PROGRAM StructuredText
VAR
	ChangeTime		:TIME:=T#1S;
	CountOnes		:INT:=1;
	CountFives		:INT:=1;
	JustOncePer 	:R_TRIG;
	DidSomething:BOOL;
	AlsoCountTo25	: BOOL;
END_VAR
VAR CONSTANT
	ST_DURATION	:TIME:=T#2S;
END_VAR

	Comparison_GVL.DefaultOFF	:=	Comparison_GVL.NormallyOpen_NO; //Sets DefaultOFF equal to whatever NormallyOpen is set to
	Comparison_GVL.DefaultON	:=	NOT Comparison_GVL.NormallyClosed_NC; //Sets DefaultON equal to the opposite of what NormallyClosed is set to
	
	Comparison_GVL.Tada			:= Comparison_GVL.This_And AND Comparison_GVL.And_This	AND NOT Comparison_GVL.But_NOT_This	AND
								(Comparison_GVL.This_Or OR Comparison_GVL.Or_This OR NOT Comparison_GVL.Or_NOT_This);
	
	// this line ^ and this next one technically do the same thing BUT if I wanted to do more complicated stuff or multiple things I need to use the IF 
	
	IF Comparison_GVL.This_And AND Comparison_GVL.And_This	AND NOT Comparison_GVL.But_NOT_This	AND
		(Comparison_GVL.This_Or OR Comparison_GVL.Or_This OR NOT Comparison_GVL.Or_NOT_This) THEN
		Comparison_GVL.Tada	:= TRUE;
	ELSE
		Comparison_GVL.Tada	:= FALSE;
	END_IF
	
	Comparison_GVL.OffTimer_TOF(IN:=Comparison_GVL.TurnOFFAfter,PT:= ST_DURATION);
	Comparison_GVL.OnTimer_TON(IN:=Comparison_GVL.TurnONAfter,PT:= ST_DURATION);
	Comparison_GVL.PulseTimer_TP(IN:=NOT Comparison_GVL.PulseTimer_TP.Q,PT:= ChangeTime);
	JustOncePer(CLK:= Comparison_GVL.PulseTimer_TP.Q);
	
	IF JustOncePer.Q THEN
		CountOnes:= CountOnes+1;
		Comparison_GVL.TurnOnFor:=FALSE;
	END_IF
	IF CountOnes = 5 THEN
		CountFives:= CountFives +1;
		CountOnes:=1;
	END_IF	
	
	DidSomething:= DoSomething(Counter:= (CountOnes*CountFives) );
	
	IF CountFives = 5 THEN
		CountFives:=1;
	END_IF

METHOD DoSomething : BOOL
VAR_INPUT
	Counter:INT;
END_VAR
CASE Counter OF
	1,10,20:
		Comparison_GVL.TurnOFFAfter:=TRUE;
		Comparison_GVL.TurnONAfter:=TRUE;
		DoSomething:=TRUE;
	2,11,21:
		Comparison_GVL.TurnOFFAfter:=FALSE;
		DoSomething:=TRUE;
	3:
		Comparison_GVL.This_And:=TRUE;
		Comparison_GVL.And_This:=TRUE;
		DoSomething:=TRUE;
	5:
		Comparison_GVL.But_NOT_This:=FALSE;
		DoSomething:=TRUE;
	7:
		Comparison_GVL.This_Or:=TRUE;
		DoSomething:=TRUE;
	9,19:
		Comparison_GVL.TurnONAfter:=FALSE;
		DoSomething:=TRUE;
	13:
		Comparison_GVL.Or_This:=TRUE;
		DoSomething:=TRUE;
	15:
		Comparison_GVL.Or_This:=FALSE;
		Comparison_GVL.Or_NOT_This:=FALSE;
		DoSomething:=TRUE;
	17:
		Comparison_GVL.This_Or:=FALSE;
		Comparison_GVL.Or_This:=FALSE;
		DoSomething:=TRUE;
	25:
		AlsoCountTo25:=TRUE;
	ELSE
		DoSomething:=FALSE;
		Comparison_GVL.TurnOnFor:=TRUE;
END_CASE
END_METHOD

END_PROGRAM

(* stored: Version 1.1.0.1, ProductVersion 3.1.4024.11
   POU StructuredText: Id {7ea544f2-f1c6-45f3-b400-669543b4addc}, SpecialFunc None
   Method DoSomething: Id {9372d4a4-4fdc-453f-ab7c-ac838f9d2fbc} *)
